FUNCTION_BLOCK PossibilittyLogic
VAR_INPUT
	TriggerInput:BOOL;
END_VAR
VAR_OUTPUT
	TriggerOutput:BOOL;
END_VAR
VAR
	Counter:INT;
	FalseCounter:int;
	TriggerON:R_TRIG;
	TriggerOFF:F_Trig;
END_VAR


///Increment the counter when the bit is high
TriggerON(CLK:=TriggerInput,q=>);
IF TriggerON.Q THEN
  TriggerOutput:=TRUE;
  FalseCounter:=0;
END_IF
///Decrement the counter when the bit is low
//Increment the countier if the input is continoussly low
IF TriggerInput=FALSE THEN
   FalseCounter:=FalseCounter+1;
   IF  FalseCounter>1000 THEN
	   falseCounter:=0;
   END_IF
END_IF

IF FalseCounter>700 THEN
   TriggerOutput:=FALSE;   
   END_IF

END_FUNCTION_BLOCK

(* stored: Version 1.1.0.1, ProductVersion 3.1.4022.16
   POU PossibilittyLogic: Id {2e7537d5-03e3-48af-bf65-1054c43925b2}, SpecialFunc None *)
